// TIA Portal V19 export
VAR_GLOBAL   // PLC tag table "D02"
   D02_Ls AT %I1020.1 : Bool;   // 102DI1 - 190SQ1
END_VAR
